FUNCTION_BLOCK FB_UPS_CU81x0_0xx0 EXTENDS FB_UPS_Base
VAR_INPUT
END_VAR
VAR_OUTPUT
END_VAR
VAR
	fbUps			:FB_GetUPSStatus;
	_stUpsStatus	:ST_UPSStatus;
END_VAR

METHOD Execute
fbUps(	sNetId		:=SUPER^._PcAmsNetId,
		nPort		:=0,
		bEnable		:=TRUE,
		bValid		=>,
		bError		=>,
		nErrId		=>,
		stStatus	=>_stUpsStatus
		);

SUPER^._bReady:= fbUps.stStatus.ePowerStatus=E_UpsPowerStatus.PowerOnLine;

SUPER^._bPowerFailDetect:= fbUps.stStatus.ePowerStatus=E_UpsPowerStatus.PowerOnBattery;

SUPER^._bReplaceBattery:=fbUps.stStatus.eBatteryStatus=E_BatteryStatus.BatteryReplace;

SUPER^._nBatteryPercent:=fbUps.stStatus.BatteryLifePercent;
END_METHOD

PROPERTY stUpsStatus : ST_UPSStatus
GET
stUpsStatus:=_stUpsStatus;
END_GET
END_PROPERTY

END_FUNCTION_BLOCK

(* stored: Version 1.1.0.1
   POU FB_UPS_CU81x0_0xx0: Id {1271138a-62b6-4969-8bf3-f7871e338543}, SpecialFunc None
   Method Execute: Id {e8864bcd-5c89-408c-b4fe-4b644cc2d5e6}
   Property stUpsStatus: Id {13aa49ed-cf01-4f0e-9e2f-17c41c8576c9}
   Get Get: Id {c05dad3e-48b0-4e49-8e3c-8a0ba4108add} *)
